(* IEC 61131-3 sources: ae-tiax/test/TrafficLight, 4 files *)

(* ---- TestStateGreen.st ---- *)
USING Simatic.Ax.Tiax;
USING AxUnit.Assert;
NAMESPACE Simatic.Ax.TrafficLight
    {TestFixture}
    CLASS TestStateGreen
        VAR PUBLIC
            state : StateGreen;
            light : BOOL;
        END_VAR

        {Test}
        METHOD PUBLIC OnEntry_switch_on_green_light
            state.gn := REF(light);
            state.OnEntry();
            Equal(expected := TRUE, actual := light);
        END_METHOD

        {Test}
        METHOD PUBLIC OnEntry_counts_the_activations
            Equal(expected := 0, actual := state.GetActivations());
            THIS.OnEntry_switch_on_green_light();
            Equal(expected := 1, actual := state.GetActivations());
        END_METHOD

        {Test}
        METHOD PUBLIC Actions_counts_each_call
            Equal(expected := 0, actual := state.GetCalls());
            state.Action();
            Equal(expected := 1, actual := state.GetCalls());
            state.Action();
            Equal(expected := 2, actual := state.GetCalls());
        END_METHOD

        {Test}
        METHOD PUBLIC OnExit_switch_off_green_light
            // first switch on the light
            THIS.OnEntry_switch_on_green_light();
            // then Call the onExit method
            state.OnExit();
            Equal(expected := FALSE, actual := light);
        END_METHOD
        {Test}
        METHOD PUBLIC GetColor_returns_green
            Equal(expected := TRUE, actual := state.GetColor() = Colors#Green);
        END_METHOD

    END_CLASS
END_NAMESPACE

(* ---- TestStateRed.st ---- *)
USING Simatic.Ax.Tiax;
USING AxUnit.Assert;
NAMESPACE Simatic.Ax.TrafficLight
    {TestFixture}
    CLASS TestStateRed
        VAR PUBLIC
            state : StateRed;
            light : BOOL;
        END_VAR

        {Test}
        METHOD PUBLIC OnEntry_switch_on_red_light
            state.rd := REF(light);
            state.OnEntry();
            Equal(expected := TRUE, actual := light);
        END_METHOD

        {Test}
        METHOD PUBLIC OnEntry_counts_the_activations
            Equal(expected := 0, actual := state.GetActivations());
            THIS.OnEntry_switch_on_red_light();
            Equal(expected := 1, actual := state.GetActivations());
        END_METHOD

        {Test}
        METHOD PUBLIC Actions_counts_each_call
            Equal(expected := 0, actual := state.GetCalls());
            state.Action();
            Equal(expected := 1, actual := state.GetCalls());
            state.Action();
            Equal(expected := 2, actual := state.GetCalls());
        END_METHOD

        {Test}
        METHOD PUBLIC OnExit_switch_off_red_light
            // first switch on the light
            THIS.OnEntry_switch_on_red_light();
            // then Call the onExit method
            state.OnExit();
            Equal(expected := FALSE, actual := light);
        END_METHOD
        {Test}
        METHOD PUBLIC GetColor_returns_red
            Equal(expected := TRUE, actual := state.GetColor() = Colors#Red);
        END_METHOD

    END_CLASS
END_NAMESPACE

(* ---- TestStateRedYellow.st ---- *)
USING AxUnit.Assert;
USING Simatic.Ax.Tiax;
NAMESPACE Simatic.Ax.TrafficLight
    {TestFixture}
    CLASS TestStateRedYellow
        VAR PUBLIC
            state : StateRedYellow;
            lightYellow : BOOL;
            lightRed : BOOL;
        END_VAR

        {Test}
        METHOD PUBLIC OnEntry_switch_on_red_yellow_light
            state.ye := REF(lightYellow);
            state.rd := REF(lightRed);
            state.OnEntry();
            Equal(expected := TRUE, actual := lightYellow);
            Equal(expected := TRUE, actual := lightRed);
        END_METHOD

        {Test}
        METHOD PUBLIC OnEntry_counts_the_activations
            Equal(expected := 0, actual := state.GetActivations());
            THIS.OnEntry_switch_on_red_yellow_light();
            Equal(expected := 1, actual := state.GetActivations());
        END_METHOD

        {Test}
        METHOD PUBLIC Actions_counts_each_call
            Equal(expected := 0, actual := state.GetCalls());
            state.Action();
            Equal(expected := 1, actual := state.GetCalls());
            state.Action();
            Equal(expected := 2, actual := state.GetCalls());
        END_METHOD

        {Test}
        METHOD PUBLIC OnExit_switch_off_red_yellow_light
            // first switch on the light
            THIS.OnEntry_switch_on_red_yellow_light();
            // then Call the onExit method
            state.OnExit();
            Equal(expected := FALSE, actual := lightYellow);
            Equal(expected := FALSE, actual := lightRed);
        END_METHOD
        {Test}
        METHOD PUBLIC GetColor_returns_red_yellow
            Equal(expected := TRUE, actual := state.GetColor() = Colors#RED_YELLOW);
        END_METHOD

    END_CLASS
END_NAMESPACE

(* ---- TestStateYellow.st ---- *)
USING AxUnit.Assert;
USING Simatic.Ax.Tiax;
NAMESPACE Simatic.Ax.TrafficLight
    {TestFixture}
    CLASS TestStateYellow
        VAR PUBLIC
            state : StateYellow;
            light : BOOL;
        END_VAR

        {Test}
        METHOD PUBLIC OnEntry_switch_on_yellow_light
            state.ye := REF(light);
            state.OnEntry();
            Equal(expected := TRUE, actual := light);
        END_METHOD

        {Test}
        METHOD PUBLIC OnEntry_counts_the_activations
            Equal(expected := 0, actual := state.GetActivations());
            THIS.OnEntry_switch_on_yellow_light();
            Equal(expected := 1, actual := state.GetActivations());
        END_METHOD

        {Test}
        METHOD PUBLIC Actions_counts_each_call
            Equal(expected := 0, actual := state.GetCalls());
            state.Action();
            Equal(expected := 1, actual := state.GetCalls());
            state.Action();
            Equal(expected := 2, actual := state.GetCalls());
        END_METHOD

        {Test}
        METHOD PUBLIC OnExit_switch_off_yellow_light
            // first switch on the light
            THIS.OnEntry_switch_on_yellow_light();
            // then Call the onExit method
            state.OnExit();
            Equal(expected := FALSE, actual := light);
        END_METHOD
        {Test}
        METHOD PUBLIC GetColor_returns_yellow
            Equal(expected := TRUE, actual := state.GetColor() = Colors#Yellow);
        END_METHOD

    END_CLASS
END_NAMESPACE
